// SIMATIC S7-200 SMART project (STEP 7-Micro/WIN SMART), CPU ST40

SYMBOL_TABLE 系统符号
Clock_1s         SM0.5    // 针对 1 s 的周期时间，时钟脉冲接通 0.5 s，断开 0.5 s.
END_SYMBOL_TABLE

ORGANIZATION_BLOCK MAIN:OB1
TITLE=程序注释
BEGIN
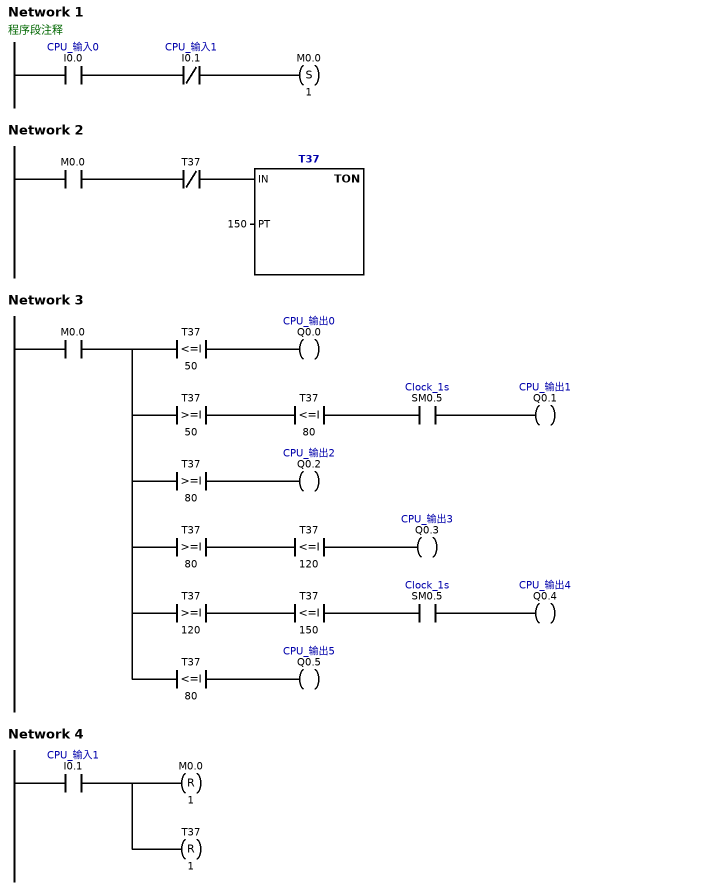
Network 1
// 程序段注释
// (network saved uncompiled; LAD cells follow)
// row 0: c0 -| |- CPU_输入0:I0.0  c1 -|/|- CPU_输入1:I0.1  c2 -(S) M0.0, 1
Network 2
// (network saved uncompiled; LAD cells follow)
// row 0: c0 -| |- M0.0  c1 -|/|- T37  c2 [TON T37 IN:=power@row0, PT:=150]
// row 1: c2 [box]
Network 3
// (network saved uncompiled; LAD cells follow)
// row 0: c0 -| |- M0.0 v  c1 -|<=I|- T37, 50  c2 -( ) CPU_输出0:Q0.0
// row 1: c0 ^v  c1 -|>=I|- T37, 50  c2 -|<=I|- T37, 80  c3 -| |- Clock_1s:SM0.5  c4 -( ) CPU_输出1:Q0.1
// row 2: c0 ^v  c1 -|>=I|- T37, 80  c2 -( ) CPU_输出2:Q0.2
// row 3: c0 ^v  c1 -|>=I|- T37, 80  c2 -|<=I|- T37, 120  c3 -( ) CPU_输出3:Q0.3
// row 4: c0 ^v  c1 -|>=I|- T37, 120  c2 -|<=I|- T37, 150  c3 -| |- Clock_1s:SM0.5  c4 -( ) CPU_输出4:Q0.4
// row 5: c0 ^  c1 -|<=I|- T37, 80  c2 -( ) CPU_输出5:Q0.5
Network 4
// (network saved uncompiled; LAD cells follow)
// row 0: c0 -| |- CPU_输入1:I0.1 v  c1 -(R) M0.0, 1
// row 1: c0 ^  c1 -(R) T37, 1
END_ORGANIZATION_BLOCK
